Fanuc KAREL source: kb00127.KL

-- PROVISIONAL review KL for V770-1; original PC SHA256 b44d6688c82ce412850fb8f641eaca7ebbcbc4af471d99ecf3ef97ec5729c47c
-- Incomplete behavior may be omitted. Consult companion uncertainty JSON. Do not deploy.
PROGRAM KB00127
%NOLOCKGROUP
VAR
  P1 : STRING[80]
  P2 : INTEGER
  RESULT : INTEGER
BEGIN
  -- UNRESOLVED_PC offsets 5-14; opcodes 3F,75
  -- UNRESOLVED_PC offsets 19-26; opcodes 9D,23
  -- UNRESOLVED_PC offsets 31-54; opcodes 27,22,2A,22,76,23
  -- UNRESOLVED_PC offsets 59-63; opcodes 7F
END KB00127
